{attribute 'qualified_only'}
{attribute 'strict'}
TYPE Modos :
(
	Stop:=0,
	Auto,
	Manual,
	StopSec,
	Reseteando,
	Parando
);
END_TYPE

(* stored: Version 1.1.0.1, ProductVersion 3.1.4024.9
   DUT Modos: Id {4fbbaf29-9476-4dfd-a35c-75706e7665d7} *)
